// TIA Portal V19 export
FUNCTION "Straightener_CALL" : Void   // FC123, LAD
TITLE = STRAIGHTENER CALL
// stored: SetENOAutomatically false
   VAR_TEMP
      i : Int;
   END_VAR
BEGIN

REGION Network 1: Data In - PB Feed
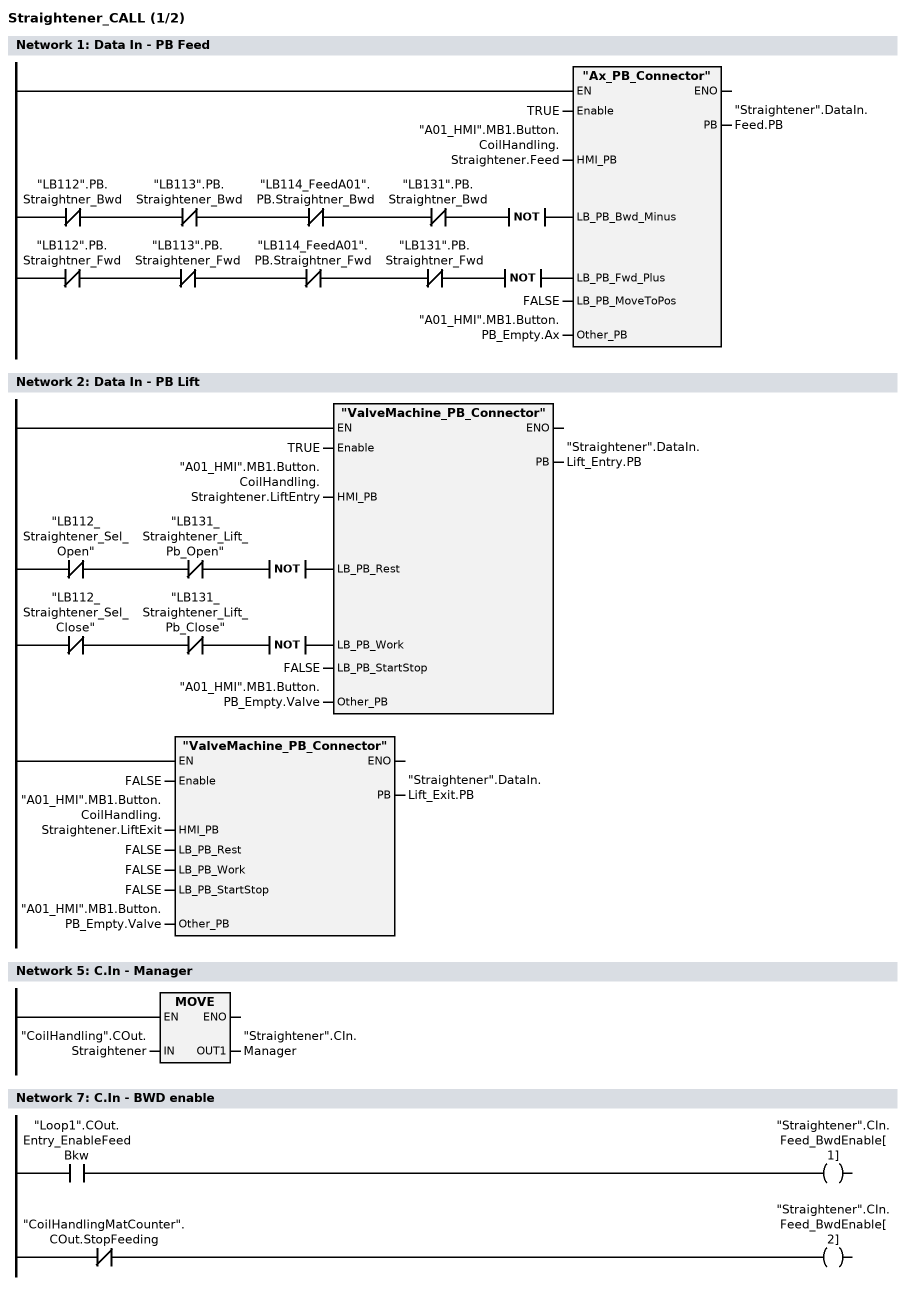
   RUNG wire#powerrail
      "Ax_PB_Connector"(LB_PB_Bwd_Minus := wire#w1, LB_PB_Fwd_Plus := wire#w2, Enable := TRUE, HMI_PB := "A01_HMI".MB1.Button.CoilHandling.Straightener.Feed, LB_PB_MoveToPos := FALSE, Other_PB := "A01_HMI".MB1.Button.PB_Empty.Ax, PB => "Straightener".DataIn.Feed.PB)
   END_RUNG
   RUNG wire#powerrail
      I_Contact( "LB112".PB.Straightner_Bwd )
      I_Contact( "LB113".PB.Straightener_Bwd )
      I_Contact( "LB114_FeedA01".PB.Straightner_Bwd )
      I_Contact( "LB131".PB.Straightner_Bwd )
      Not()
   END_RUNG wire#w1
   RUNG wire#powerrail
      I_Contact( "LB112".PB.Straightner_Fwd )
      I_Contact( "LB113".PB.Straightener_Fwd )
      I_Contact( "LB114_FeedA01".PB.Straightner_Fwd )
      I_Contact( "LB131".PB.Straightner_Fwd )
      Not()
   END_RUNG wire#w2
   // the same network as SCL:
   "Ax_PB_Connector"(Enable := TRUE,
                     HMI_PB := "A01_HMI".MB1.Button.CoilHandling.Straightener.Feed,
                     LB_PB_Bwd_Minus := NOT (NOT "LB112".PB.Straightner_Bwd AND NOT "LB113".PB.Straightener_Bwd AND NOT "LB114_FeedA01".PB.Straightner_Bwd AND NOT "LB131".PB.Straightner_Bwd),
                     LB_PB_Fwd_Plus := NOT (NOT "LB112".PB.Straightner_Fwd AND NOT "LB113".PB.Straightener_Fwd AND NOT "LB114_FeedA01".PB.Straightner_Fwd AND NOT "LB131".PB.Straightner_Fwd),
                     LB_PB_MoveToPos := FALSE,
                     Other_PB := "A01_HMI".MB1.Button.PB_Empty.Ax,
                     PB => "Straightener".DataIn.Feed.PB);
END_REGION

REGION Network 2: Data In - PB Lift
   RUNG wire#powerrail
      "ValveMachine_PB_Connector"(LB_PB_Rest := wire#w1, LB_PB_Work := wire#w2, Enable := TRUE, HMI_PB := "A01_HMI".MB1.Button.CoilHandling.Straightener.LiftEntry, LB_PB_StartStop := FALSE, Other_PB := "A01_HMI".MB1.Button.PB_Empty.Valve, PB => "Straightener".DataIn.Lift_Entry.PB)
   END_RUNG
   RUNG wire#powerrail
      I_Contact( "LB112_Straightener_Sel_Open" )
      I_Contact( "LB131_Straightener_Lift_Pb_Open" )
      Not()
   END_RUNG wire#w1
   RUNG wire#powerrail
      I_Contact( "LB112_Straightener_Sel_Close" )
      I_Contact( "LB131_Straightener_Lift_Pb_Close" )
      Not()
   END_RUNG wire#w2
   RUNG wire#powerrail
      "ValveMachine_PB_Connector"(Enable := FALSE, HMI_PB := "A01_HMI".MB1.Button.CoilHandling.Straightener.LiftExit, LB_PB_Rest := FALSE, LB_PB_Work := FALSE, LB_PB_StartStop := FALSE, Other_PB := "A01_HMI".MB1.Button.PB_Empty.Valve, PB => "Straightener".DataIn.Lift_Exit.PB)
   END_RUNG
   // the same network as SCL:
   "ValveMachine_PB_Connector"(Enable := TRUE,
                           HMI_PB := "A01_HMI".MB1.Button.CoilHandling.Straightener.LiftEntry,
                           LB_PB_Rest := NOT (NOT "LB112_Straightener_Sel_Open" AND NOT "LB131_Straightener_Lift_Pb_Open"),
                           LB_PB_Work := NOT (NOT "LB112_Straightener_Sel_Close" AND NOT "LB131_Straightener_Lift_Pb_Close"),
                           LB_PB_StartStop := FALSE,
                           Other_PB := "A01_HMI".MB1.Button.PB_Empty.Valve,
                           PB => "Straightener".DataIn.Lift_Entry.PB);
   "ValveMachine_PB_Connector"(Enable := FALSE,
                           HMI_PB := "A01_HMI".MB1.Button.CoilHandling.Straightener.LiftExit,
                           LB_PB_Rest := FALSE,
                           LB_PB_Work := FALSE,
                           LB_PB_StartStop := FALSE,
                           Other_PB := "A01_HMI".MB1.Button.PB_Empty.Valve,
                           PB => "Straightener".DataIn.Lift_Exit.PB);
END_REGION

REGION Network 3 (SCL): Data In - Sensori

   //Feed
   "Straightener".DataIn.Feed.Fan_M_Feedback := "Straightener_MotorFan_FdbkKM";

   // Lift entry
   "Straightener".DataIn.Lift_Entry.Rest_Ls[1] := "Raddrizzatrice_Ls_Rullo_Aperto";
END_REGION

REGION Network 4: >
END_REGION

REGION Network 5: C.In - Manager
   RUNG wire#powerrail
      Move(in := "CoilHandling".COut.Straightener, out1 => "Straightener".CIn.Manager)
   END_RUNG
   // the same network as SCL:
   "Straightener".CIn.Manager := "CoilHandling".COut.Straightener;
END_REGION

REGION Network 6 (SCL): CIn - Init BWD & FWD enable
   FOR #i := 1 TO 8 DO

       "Straightener".CIn.Feed_BwdEnable[#i] := TRUE;
       "Straightener".CIn.Feed_FwdEnable[#i] := TRUE;
   END_FOR;
END_REGION

REGION Network 7: C.In - BWD enable
   RUNG wire#powerrail
      Contact( "Loop1".COut.Entry_EnableFeedBkw )
      Coil( "Straightener".CIn.Feed_BwdEnable[1] )
   END_RUNG
   RUNG wire#powerrail
      I_Contact( "CoilHandlingMatCounter".COut.StopFeeding )
      Coil( "Straightener".CIn.Feed_BwdEnable[2] )
   END_RUNG
   // the same network as SCL:
   "Straightener".CIn.Feed_BwdEnable[1] := "Loop1".COut.Entry_EnableFeedBkw;
   "Straightener".CIn.Feed_BwdEnable[2] := NOT "CoilHandlingMatCounter".COut.StopFeeding;
END_REGION

REGION Network 8: C.In - FWD enable
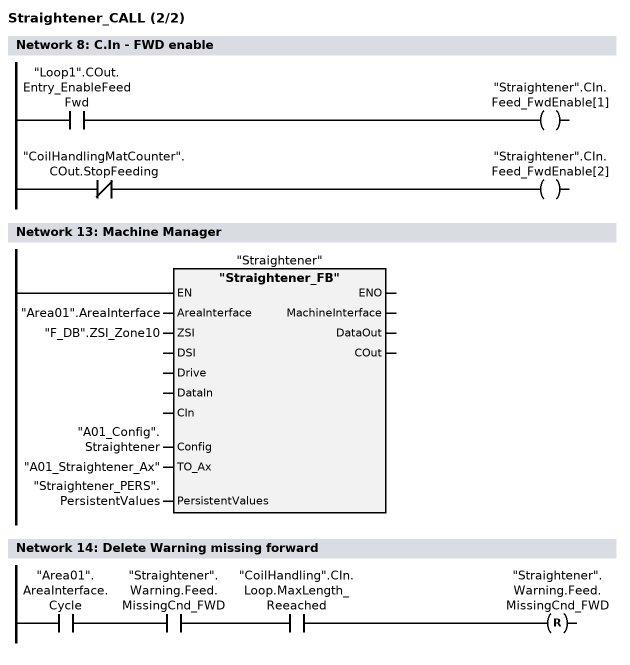
   RUNG wire#powerrail
      Contact( "Loop1".COut.Entry_EnableFeedFwd )
      Coil( "Straightener".CIn.Feed_FwdEnable[1] )
   END_RUNG
   RUNG wire#powerrail
      I_Contact( "CoilHandlingMatCounter".COut.StopFeeding )
      Coil( "Straightener".CIn.Feed_FwdEnable[2] )
   END_RUNG
   // the same network as SCL:
   "Straightener".CIn.Feed_FwdEnable[1] := "Loop1".COut.Entry_EnableFeedFwd;
   "Straightener".CIn.Feed_FwdEnable[2] := NOT "CoilHandlingMatCounter".COut.StopFeeding;
END_REGION

REGION Network 9: >
END_REGION

REGION Network 10 (SCL): DSI
   "Straightener".DSI.Feed := "F_DB".DSI_S120_Straightener;

   "Straightener".DSI.Lift_Entry :=
   "Straightener".DSI.Lift_Exit := "F_DB".DSI_V_Air_Gen;
END_REGION

REGION Network 11 (SCL): Drive
   "Straightener".Drive.Feed.Infeed_ON := "Areas_ITF".AG.Infeed_Running;
   "Straightener".Drive.Feed.AccessPoint := "HW_Const_Values".CU2_PN_830A1_ModuleAccessPoint;
   "Straightener".Drive.Feed.AxisID := "CU2_ID_4_830A1_830M1";
   "Straightener".Drive.Feed.TokenChain := "TOKENCHAIN_CU2";
END_REGION

REGION Network 12: >
END_REGION

REGION Network 13: Machine Manager
   RUNG wire#powerrail
      "Straightener"(AreaInterface := "Area01".AreaInterface, ZSI := "F_DB".ZSI_Zone10, DSI :=, Drive :=, DataIn :=, CIn :=, Config := "A01_Config".Straightener, TO_Ax := "A01_Straightener_Ax", PersistentValues := "Straightener_PERS".PersistentValues, MachineInterface =>, DataOut =>, COut =>)
   END_RUNG
   // the same network as SCL:
   "Straightener"(AreaInterface := "Area01".AreaInterface,   // "Straightener_FB"
                  ZSI := "F_DB".ZSI_Zone10,
                  Config := "A01_Config".Straightener,
                  TO_Ax := "A01_Straightener_Ax",
                  PersistentValues := "Straightener_PERS".PersistentValues);
END_REGION

REGION Network 14: Delete Warning missing forward
   RUNG wire#powerrail
      Contact( "Area01".AreaInterface.Cycle )
      Contact( "Straightener".Warning.Feed.MissingCnd_FWD )
      Contact( "CoilHandling".CIn.Loop.MaxLength_Reeached )
      R_Coil( "Straightener".Warning.Feed.MissingCnd_FWD )
   END_RUNG
   // the same network as SCL:
   IF "Area01".AreaInterface.Cycle AND "Straightener".Warning.Feed.MissingCnd_FWD AND "CoilHandling".CIn.Loop.MaxLength_Reeached THEN
       "Straightener".Warning.Feed.MissingCnd_FWD := FALSE;
   END_IF;
END_REGION

REGION Network 15: >
END_REGION

REGION Network 16 (SCL): Data Out
   "Straightener_MotorFan_KM" := "Straightener".DataOut.Feed.Fan_M_Contactor;

   //Lift Entry
   "Straightener_LiftEntry_V_Open" := "Straightener".DataOut.Lift_Entry.RestSolenoid;
   "Straightener_LiftEntry_V_Close" := "Straightener".DataOut.Lift_Entry.WorkSolenoid;

   (*
   //Lift Exit
   "Straightener_LiftExit_V_Open" := "Straightener".DataOut.Lift_Exit.RestSolenoid;
   "Straightener_LiftExit_V_Close" := "Straightener".DataOut.Lift_Exit.WorkSolenoid;
   *)
END_REGION

REGION Network 17: >
END_REGION

REGION Network 18: >
END_REGION

REGION Network 19: >
END_REGION
END_FUNCTION
